FUNCTION_BLOCK BeltConveyor EXTENDS Conveyor
VAR_INPUT
END_VAR
VAR_OUTPUT
END_VAR
VAR
END_VAR

Super^();

END_FUNCTION_BLOCK

(* stored: Version 1.1.0.1, ProductVersion 3.1.4024.2
   POU BeltConveyor: Id {72c43a83-ea83-4506-b00d-047ee4dbd58a}, SpecialFunc None *)
